{attribute addProperty BoxType "ATH2050-5501-0022"}
{attribute addProperty Id "BinaryDataAT %I*ARRAY [0..55] OF BYTE00"}
{attribute addProperty CRC "916431119"}
{attribute addProperty SizeInBites "0"}
{attribute addProperty SizeInBytes "0"}
TYPE FB_Inputs_369FA10F :
STRUCT
	{attribute addProperty Name "BinaryData"}
	BinaryData AT %I* : ARRAY [0..55] OF BYTE;
END_STRUCT
END_TYPE

(* stored: Version 1.2.0.0, ProductVersion 3.1.4024.9
   DUT FB_Inputs_369FA10F: Id {ee163a3d-2a9f-49cb-9a31-49bdfd4c2c64} *)
